{attribute 'GeneratedUsingTerminal: EL3311-0000-0018'}
{attribute addProperty BoxType "EL3311-0000-0018"}
{attribute addProperty Description "EL3311 1Ch. Ana. Input Thermocouple (TC)"}
{attribute addProperty Physics "KK"}
{attribute addProperty Id "TC_InputsAT %I*AI_Standard_Channel_4A3944819WcStateAT %I*WcState_9091E0EB2InfoDataAT %I*InfoData_32EB74EA10"}
{attribute addProperty CRC "413671248"}
{attribute addProperty Size "21"}
TYPE EL3311_18A81F50 EXTENDS EtcSlaveTerminalBase_947E5A46 :
STRUCT
	{attribute addProperty Name "TC_Inputs"}
	TC_Inputs : AI_Standard_Channel_4A394481;
	{attribute addProperty Name "WcState"}
	WcState : WcState_9091E0EB;
	{attribute addProperty Name "InfoData"}
	InfoData : InfoData_32EB74EA;
END_STRUCT
END_TYPE

(* stored: Version 1.2.0.0, ProductVersion 3.1.4024.9
   DUT EL3311_18A81F50: Id {d2fdbe05-7f42-4a82-bf2d-24c5d86a0520} *)
